FUNCTION_BLOCK LGCS_MAIN_CONTROLLER (* Basic FB with empty ECC *)
  (* Standard: 61499-2 *)
  (* Version 1.0, 2022-01-11, Fan *)
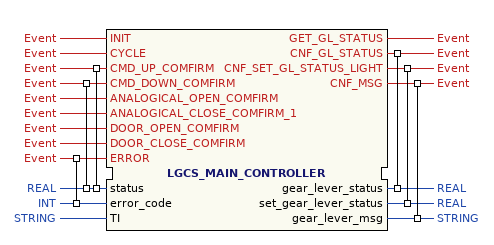
  EVENT_INPUT
    INIT;
    CYCLE;
    CMD_UP_COMFIRM WITH status;
    CMD_DOWN_COMFIRM WITH status;
    ANALOGICAL_OPEN_COMFIRM;
    ANALOGICAL_CLOSE_COMFIRM_1;
    DOOR_OPEN_COMFIRM;
    DOOR_CLOSE_COMFIRM;
    ERROR WITH error_code;
  END_EVENT
  EVENT_OUTPUT
    GET_GL_STATUS;
    CNF_GL_STATUS WITH gear_lever_status;
    CNF_SET_GL_STATUS_LIGHT WITH set_gear_lever_status;
    CNF_MSG WITH gear_lever_msg;
  END_EVENT
  VAR_INPUT
    status : REAL;
    error_code : INT;
    TI : STRING;
  END_VAR
  VAR_OUTPUT
    gear_lever_status : REAL;
    set_gear_lever_status : REAL;
    gear_lever_msg : STRING;
  END_VAR
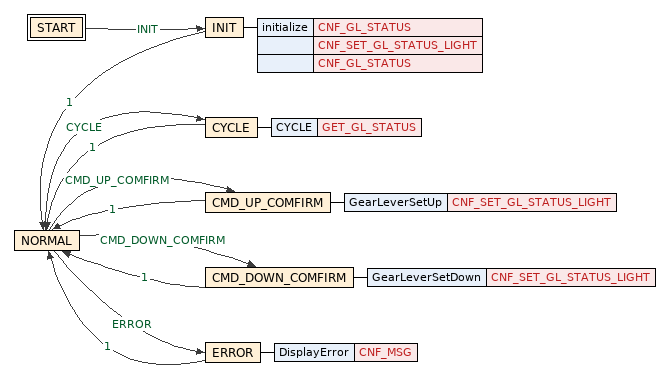
  EC_STATES
    START; (* Initial State *)
    NORMAL;
    INIT : initialize -> CNF_GL_STATUS, -> CNF_SET_GL_STATUS_LIGHT, -> CNF_GL_STATUS;
    CYCLE : CYCLE -> GET_GL_STATUS;
    CMD_UP_COMFIRM : GearLeverSetUp -> CNF_SET_GL_STATUS_LIGHT;
    CMD_DOWN_COMFIRM : GearLeverSetDown -> CNF_SET_GL_STATUS_LIGHT;
    ERROR : DisplayError -> CNF_MSG;
  END_STATES
  EC_TRANSITIONS
    START TO INIT := INIT;
    INIT TO NORMAL := 1;
    NORMAL TO CYCLE := CYCLE;
    CYCLE TO NORMAL := 1;
    NORMAL TO CMD_UP_COMFIRM := CMD_UP_COMFIRM;
    CMD_UP_COMFIRM TO NORMAL := 1;
    NORMAL TO CMD_DOWN_COMFIRM := CMD_DOWN_COMFIRM;
    CMD_DOWN_COMFIRM TO NORMAL := 1;
    NORMAL TO ERROR := ERROR;
    ERROR TO NORMAL := 1;
  END_TRANSITIONS
  ALGORITHM initialize IN AnyText: (* Initialization algorithm *)
	cout << "[LGCS_MAIN_CONTROLLER1] alg_initialize()\n";
	// Set default the Gear lever status
	gear_lever_status() = false;
  END_ALGORITHM
  ALGORITHM CYCLE IN AnyText: (* Cycle controller *)

  END_ALGORITHM
  ALGORITHM GearLeverSetUp IN AnyText: (* Gear lever set up *)
	cout << "[Z_CONTROLLER2] alg_SetUp\n"
	SET_TEMP() = SET_TEMP();
  END_ALGORITHM
  ALGORITHM GearLeverSetDown IN AnyText: (* Gear lever set down *)
	cout << "[Z_CONTROLLER2] alg_SetDown\n"
	SET_TEMP() = SET_TEMP();
  END_ALGORITHM
  ALGORITHM DisplayError IN AnyText: (* Report error *)

  END_ALGORITHM
END_FUNCTION_BLOCK
